// TIA Portal V20 export
// export: Created 2026-07-16T13:01:15.5465381Z, ExportSetting WithDefaults, DisplayName Totally Integrated Automation Portal, DisplayVersion V20 Update 5, DisplayName TIA Portal Openness, DisplayVersion V20 Update 4, DisplayName TIA Portal Version Control Interface, DisplayVersion V20 Update 5, DisplayName SINAMICS Startdrive Advanced, DisplayVersion V20, DisplayName SINAMICS DCC, DisplayVersion V20, DisplayName SINAMICS Startdrive G130, G150, S120, S150, SINAMICS MV, G220, S200, S210, DisplayVersion V20, DisplayName SINAMICS Startdrive G110M, G120, G120C, G120D, G120P, G115D, DisplayVersion V20, DisplayName STEP 7 Professional, DisplayVersion V20 Update 5, DisplayName STEP 7 Safety, DisplayVersion V20 Update 2, DisplayName WinCC Basic/Comfort/Advanced, DisplayVersion V20 Update 5, DisplayName WinCC Unified, DisplayVersion V20 Update 5
TYPE "MotorFwdRevIOSet"
// stored: IsFailsafeCompliant false
   STRUCT
      InHand : Bool;
      AutoStartSignal : Bool;
      HandStartSignal : Bool;
      RunningFBFwd : Bool;
      RunningFBRev : Bool;
      FaultFB : Bool;
      SystemHealthy : Bool;
      PreStartDone : Bool;
      InhibitMotor : Bool;
      FaultReset : Bool;
      FTTime : Real;
      EnableUPSTime : Real;
      FaultActive : Bool;
      RunFwd : Bool;
      RunRev : Bool;
      UPSEnable : Bool;
      FTR : Bool;
      FTS : Bool;
      HrsRun : UDInt;
      Telemetry : Int;
      Alarm : Word;
      "Name" : String;
      HandIntervention : Bool;
      RecentStart : Bool;
      TryRunMotor : Bool;
      Shutdown : Bool;
      ShutdownComplete : Bool;
      ShutdownTime : Real;
      StopMotor : Bool;
      ReverseDelay : Real;
      ReverseIgnoreFT : Real;
      Reverse : Bool;
      HandReverse : Bool;
   END_STRUCT;
END_TYPE
